// TwinCAT 3 PLC project Crane_Control
// ProgramVersion: 3.1.4026.20
// libraries:
//   Tc2_Standard, * (Beckhoff Automation GmbH)
//   Tc2_System, * (Beckhoff Automation GmbH)
// project tree:
//   Enumeration/ E_Mode.TcDUT (not stored), E_Motion.TcDUT (not stored)
//   Function Blocks/ FB_AutoClock.TcPOU, FB_ControlSignal.TcPOU, FB_Derivator.TcPOU (not stored), FB_FeedForward.TcPOU, FB_FeedForward_NonLinear.TcPOU, FB_Filtering.TcPOU, FB_Home.TcPOU, FB_InitialPos.TcPOU, FB_Integrator.TcPOU, FB_JoystickInputScaling.TcPOU, FB_KvFF.TcPOU (not stored), FB_MotionRef.TcPOU, FB_NaiveFF.TcPOU, FB_Normalize.TcPOU (not stored), FB_PID.TcPOU, FB_PositionInputScaling.TcPOU (not stored), FB_PressureFeedback.TcPOU, FB_RunClock.TcPOU (not stored), FB_Running.TcPOU, FB_ValveOutput.TcPOU (not stored)
//   Global Variable Lists/ G_Enables.TcGVL, G_FilterConstants.TcGVL (not stored), G_Filtered.TcGVL (not stored), G_Init.TcGVL, G_Inputs.TcGVL (not stored), G_Mode.TcGVL (not stored), G_OPC.TcGVL, G_Output.TcGVL, G_Parameter.TcGVL
//   / PlcTask.TcTTO
//   Programs/ MAIN.TcPOU, P_Modes.TcPOU, P_Output.TcPOU, P_RunClock.TcPOU (not stored)
// real-time tasks:
//   TASK PlcTask: cycle T#1ms, priority 20, ADS port 350
// I/O:
//   DEVICE Device 1 (EtherCAT), AmsNetId 192.168.0.204.4.1
//     RIO (EK1100) [EK1100 EtherCAT Coupler (2A E-Bus)]
//       DI (EL1008) [EL1008 8Ch. Dig. Input 24V, 3ms]
//       DO (EL2008) [EL2008 8Ch. Dig. Output 24V, 0.5A]
//       AI1 (EL3068) [EL3068 8Ch. Ana. Input 0-10V]
//       AI2 (EL3068) [EL3068 8Ch. Ana. Input 0-10V]
//       AI3 (EL3174) [EL3174 4Ch. Ana. Input +/-10V Diff., +/-20mA SingleEnded, 16 Bit]
//       AO (EL4104) [EL4104 4Ch. Ana. Output 0-10V, 16bit]
//       End Cap (EL9011) [EL9011 End Terminal]
// variable links:
//   Crane_Control/Crane_Control Instance <-> Device 1 (EtherCAT)/RIO (EK1100)/AI2 (EL3068)
//     PlcTask Inputs/G_Inputs.nRawPs <-> AI Standard Channel 1/Value

CONFIGURATION Crane_Control
    RESOURCE PLC ON TwinCAT3
        TASK PlcTask(INTERVAL := T#10ms, PRIORITY := 20);
        PROGRAM MAIN WITH PlcTask : MAIN;
    END_RESOURCE
END_CONFIGURATION

// ---- Global Variable Lists/G_Enables.TcGVL
{attribute 'qualified_only'}
// BOOL: True/False

VAR_GLOBAL
	
	// Control Enables
	bEnablePID 		: BOOL; // Enable PID Control
	bEnableFF 		: BOOL; // Enable FeedForward	
	bEnablePFB		: BOOL; // Enable Pressure Feedback
	bEnableU 		: BOOL; // Enable Signal to Valve

	bCharTesting	: BOOL; // Enable Characteristic testing
	bMove2Home		: BOOL; // Enable Home-function
	
	// No Function
	bEnableComp 	: BOOL; // Driving with Compensator
	
	// Enumerators
	nModeSelect		: E_Motion; // Motion Reference
	
END_VAR

// ---- Global Variable Lists/G_Init.TcGVL
// SINT: Integer [-128, 127]
VAR_GLOBAL CONSTANT
	SS_INITIALIZE: SINT := 0; 	// Initial system state value
	SS_STEP: SINT := 1;			// Step sequence state value
END_VAR

// ---- Global Variable Lists/G_OPC.TcGVL
{attribute 'qualified_only'}
// LREAL: Long Real decimal number

VAR_GLOBAL
	
	// Unfiltered Pressures
	fPa 				: LREAL; // [bar], Pressure A 
	fPb 				: LREAL; // [bar], Pressure B 
	fPs 				: LREAL; // [bar], Pressure Supply 
	fPaLower 			: LREAL; // [bar], Pressure A between DCV and CBV 
	
	// Filtered Pressures
	fPaFiltered 		: LREAL; // [bar], Pressure A Filtered 
	fPbFiltered 		: LREAL; // [bar], Pressure B Filtered
	fPsFiltered 		: LREAL; // [bar], Pressure Supply Filtered
	fPaLowerFiltered 	: LREAL; // [bar], Pressure A between DCV and CBV Filtered
	
	fSpoolPosition 		: LREAL; // [-1,1], Spool position
	fPistonPosition 	: LREAL; // [m], Piston position
	fPistonPosMeasured 	: LREAL; // [m], Measured piston position
	fJoystick 			: LREAL; // [-1,1], Joystick signal
	fFlow 				: LREAL; // [L/min], Flow rod-side 
	fFlowCalc 			: LREAL; // [L/min], Calculated flow
	
	fXRef 				: LREAL; // [m], Position reference [m]
	fXDotRef 			: LREAL; // [m/s], Velocity reference [m/s]
	fFlowRef 			: LREAL; // [L/min], Flow reference calculated form fXDotRef
	
	fFFFlow				: LREAL; // [L/min], Flow form feed forward
	fKv					: LREAL; // Capacity factor (how much liquid a valve can let through over a set pressure drop)

	fWantedSpoolPos 	: LREAL; // [-1,1], Wanted spool position
	fUpfbGrad 			: LREAL; // Pressure feedback gradient
	fPxGrad 			: LREAL; // Pressure gradient
	fUTest 				: LREAL; // [-1,1], Signal to Valve with pfb (pressure feedback)
	fTime 				: LREAL; // [s], Time
	fError 				: LREAL; // [m], Error
	
	
	fSignalPID 			: LREAL; // PID signal value
	fFF 				: LREAL; // FF signal Value
	fUpfb 				: LREAL; // Pressure feedback signal
	fU 					: LREAL; // [-1,1], Signal to set spool at wanted position 

END_VAR

// ---- Global Variable Lists/G_Output.TcGVL
{attribute 'qualified_only'} // Variable needs to be used with GVL-name

// INT: [-32768, 32767]	
// BOOL: True/False
// %Q* assigns next available memory adress in Twincat (Out)

VAR_GLOBAL
	// Digital Outputs
	bGreenLight 			AT %Q* : BOOL;	// Green light on controller
	bRedLight 				AT %Q* : BOOL;	// Red light on controller
	
	// Analog Outputs
	nValveOutput 			AT %Q* : INT;	// Valve output
	bRunning				AT %Q* : BOOL;
END_VAR

// ---- Global Variable Lists/G_Parameter.TcGVL
{attribute 'qualified_only'}
// LREAL: Long Real decimal number
// INT: [-32768, 32767]	

VAR_GLOBAL
	// Motion Ref
	// Sine Parameters
	fAmplitude 		: LREAL := 0.15;
	fMean 			: LREAL := 0.2;
	fFrequency 		: LREAL := 0.05;
	
	
	// Valve Values
	// Flow
	fQMaxDown 		: LREAL := 10.0; // [L/min]
	fQMaxUp 		: LREAL := 10.0; // [L/min]	
	
	// Area
	fAreaUp 		: LREAL := 33.100/1E4; //[m^2]
	fAreaDown 		: LREAL := 23.560/1E4; //[m^2]
	
	// Deadband
	fDeadUp 		: LREAL := 0.23;
	fDeadDown 		: LREAL := 0.215;
	
	fMaxSpeed 		: LREAL := 0.01; // [m/s] 
	fDeltaP0 		: LREAL := 8.0; // [Bar]
	
	// Deadband test
	fConst 			: LREAL := 0.0; // [-1, 1]

	fCycleTime 		: LREAL := 0.001; // Time Step [s]
	fQConst 		: LREAL := 15;
	fPistonStroke 	: LREAL := 0.5;
	
	// PID-constants
	Kp 				: LREAL := 14.0; 	// P
	Ki 				: LREAL := 0.0;		// I
	Kd 				: LREAL := 0.0;		// D
	
	// Pressure feedback constants
	Kf				: LREAL := 2E-4;
	TauF			: LREAL := 0.1; // [0.05 .. 0.1]
	PFBstate		: INT 	:= 2; // 0:Switching, 1: Pa-phi*Pb, 2: Pb
	FFMode			: INT 	:= 1; // 0: Bachelor FF, 1: Kv FF, 2: Naive FF

END_VAR

// ---- Programs/MAIN.TcPOU
PROGRAM MAIN
VAR
END_VAR

P_Inputs();
P_Filtering();
P_ControlBlock();
P_Output();
//P_RunClock();
P_Modes();
P_PID();
P_FeedForward();

END_PROGRAM

// ---- Programs/P_Output.TcPOU
PROGRAM P_Output

VAR
	fbValveOutput : FB_ValveOutput;
END_VAR

// Runs FB with given values
fbValveOutput(
	fNormalizedInput := G_OPC.fU,
	bEnable := G_Enables.bEnableU,
	nOutput => G_Output.nValveOutput	
);

IF G_Mode.bRunning THEN // If system is running, set green and red light on controller true. False when not running
	G_Output.bGreenLight := TRUE;
	G_Output.bRedLight := TRUE;
ELSE
	G_Output.bGreenLight := FALSE;
	G_Output.bRedLight := FALSE;
END_IF

END_PROGRAM

// ---- Programs/P_Modes.TcPOU
PROGRAM P_Modes

VAR
	fbRunning : FB_Running;
END_VAR

// Runs FB with given values
fbRunning(
	bAuto := G_Inputs.bAuto, 			// Auto mode controller
	bManual := G_Inputs.bManual, 		// Manual mode controller
	bStart := G_Inputs.bStartButton,	// Start button
	bStop := G_Inputs.bStopButton, 		// Stop button
	
	// Values from FB sent to GVL
	bRunning => G_Mode.bRunning,
	bRunning => G_Output.bRunning,
	bManualMode => G_Mode.bManual,
	bAutoMode => G_Mode.bAuto
);

END_PROGRAM

// ---- Function Blocks/FB_Running.TcPOU
FUNCTION_BLOCK FB_Running
// BOOL: True/False

// Input variables
VAR_INPUT
	bManual : BOOL;
	bStart : BOOL;
	bStop : BOOL;
	bAuto : BOOL;
END_VAR

// Output variables
VAR_OUTPUT
	bRunning : BOOL;
	bAutoMode : BOOL;
	bManualMode : BOOL;
END_VAR


IF NOT(bStart) AND NOT(bManual) AND NOT(bAuto) OR (bStop) THEN // If nothing active, all false values
	bRunning := FALSE;
	bAutoMode := FALSE;
	bManualMode := FALSE;	
	
ELSIF bStart AND bAuto AND NOT(bStop) THEN // If start button and auto is true (auto mode)
	bRunning := TRUE;
	bAutoMode := TRUE;
	bManualMode := FALSE;
	
ELSIF bStart AND bManual AND NOT(bStop) THEN // If start and manual is true (manual mode)
	bRunning := TRUE;
	bManualMode := TRUE;
	bAutoMode := FALSE;
END_IF

END_FUNCTION_BLOCK

// ---- Function Blocks/FB_AutoClock.TcPOU
FUNCTION_BLOCK FB_AutoClock
// LREAL: Long Real decimal number
// BOOL: True/False

// Input variables
VAR_INPUT
	fStart : BOOL; // Start timer
	fRunning : BOOL; // System is running
	fCycle : LREAL; // Time step
END_VAR

// Output variables
VAR_OUTPUT
	fTime : LREAL; // Output (time)
END_VAR


IF NOT(fStart) OR NOT(fRunning) THEN // If start signal is missing or the system is not running, set time to zero
	fTime := 0.0; 
ELSIF fStart AND fRunning THEN // If both start signal and system is on. PLS ticks synced into real time
	fTime := fTime + fCycle;		
END_IF

END_FUNCTION_BLOCK

// ---- Function Blocks/FB_ControlSignal.TcPOU
FUNCTION_BLOCK FB_ControlSignal
// LREAL: Long Real decimal number
// INT: [-32768, 32767]	
// BOOL: True/False

// Input variables
VAR_INPUT
	fFF 			: LREAL; // FF signal value
	fPID			: LREAL; // PID signal value
	fPFB			: LREAL; // Pressure feedback signal
	
	// Deadband
	fDeadBandUp		: LREAL; 
	fDeadBandDown	: LREAL;
	
	nFFState		: INT; // 0: Bachelor FF, 1: Kv FF, 2: Naive FF

	bPID			: BOOL; // Enable PID control
	bFF				: BOOL; // Enable feed forward
	bPFB			: BOOL; // Enable pressure feedback
	bU				: BOOL; 
	bValve			: BOOL; 
END_VAR

// Output variables
VAR_OUTPUT
	fU				: LREAL; // Final output
	fUAdj			: LREAL; // Adjusted signal before final output
END_VAR

// Variables
VAR
	FF				: LREAL; // Feed forward
	PID				: LREAL; // PID
	PFB				: LREAL; // Pressure feedback
END_VAR


FF := fFF  * TO_INT(bFF); // Multiplies fFF with bFF. bFF:(True/False) = (1/0). Like an on/off switch for the feed forward.

PID := fPID * TO_INT(bPID); // On/off switch for PID

PFB := fPFB * TO_INT(bPFB); // On/off switch for pressure feedback

fUAdj := (FF+PID-PFB)*TO_INT(bValve); // bValve works as a main on/off switch

IF FF = 0.0 THEN // If feed forward is off
	fU := 0.0; // Output = 0
ELSE
	CASE nFFState OF // Feed forward states 0,1,2
		0: // State 0
			IF (fUAdj > 0.0) THEN
				fU := fUAdj + fDeadBandUp; // Adds offset to skip deadband in the valve (positive direction)
			ELSIF (fUAdj < 0.0) THEN
				fU := fUAdj - fDeadBandDown; // Adds offset to skip deadband in the valve (negative direction)
			ELSE
				fU := 0.0;
			END_IF
			
		ELSE // FF States that use this: 1, 2
			IF (fUAdj > 0.0) THEN
				fU := fUAdj;
			ELSIF (fUAdj < 0.0) THEN
				fU := fUAdj;
			ELSE
				fU := 0.0;
			END_IF
	END_CASE
END_IF

// Saturation for output [-1,1]
IF fU < -1.0 THEN
	fU := -1.0; 
ELSIF fU > 1.0 THEN
	fU := 1.0;
ELSE
	fU := fU;
END_IF

END_FUNCTION_BLOCK

// ---- Function Blocks/FB_FeedForward.TcPOU
FUNCTION_BLOCK FB_FeedForward
// LREAL: Long Real decimal number

// Input variables
VAR_INPUT
	fXDotRef 		: LREAL; // Velocity Reference [m/s]
	fMaxFlowUp 		: LREAL; // Needs to be positive (22)
	fMaxFlowDown 	: LREAL; // Needs to be positive (15)
	fDeadUp			: LREAL; // Needs to be positive (0.155)
	fDeadDown 		: LREAL; // Needs to be positive (0.18)
	
	fPs 			: LREAL; // [Bar]
	fPa 			: LREAL; // [Bar]
	fPb 			: LREAL; // [Bar]
	fDeltaP0		: LREAL; // [Bar] (8.0)
	fAreaUp			: LREAL; // [mm^2]
	fAreaDown		: LREAL; // [mm^2]
END_VAR

// Output variables
VAR_OUTPUT
	fUFF 			: LREAL;	// FF signal value
	fFlow			: LREAL; 	// Wanted Flow
	fFlowLM			: LREAL;	// Flow [L/min]
END_VAR

// Variables
VAR
	fDeltaP_Norm	: LREAL; 	// Pressure Drop with Compensator
	
	fDeltaP			: LREAL; 	// Pressure Drop
	fDeltaP_Ref		: LREAL; 	// Reference Pressure Drop
	fFlowRef		: LREAL; 	// Reference Flow
	
	fUFFTemp		: LREAL;	// Temp Signal Out
END_VAR


fDeltaP_Norm	:= fDeltaP0 * 100000.0; // Converts from bar to Pa

IF fXDotRef > 0.0 THEN // Velocity reference > 0
	fFlow := fXDotRef * fAreaUp; // Calculates wanted flow (Q = v*A)
	fFlowLM := -fFlow * 60000; // Converts flow to [L/min]. Negative sign for valve direction
	fDeltaP := (fPs - fPa) * 100000.0; // Calculates pressure drop
	
	IF fDeltaP < 100 THEN // Safety for pressure drop to never go below 100. Avoiding division by zero
		fDeltaP := 100;
	ELSE
		fDeltaP := fDeltaP;
	END_IF
	
	fDeltaP_Ref := ABS(fDeltaP_Norm/ (fDeltaP)); // Calculates reference pressure drop. 
	fFlowRef := (fFlow * SQRT(fDeltaP_Ref)) * 60000.0; // Calculates reference flow
	fUFFTemp := fFlowRef/fMaxFlowUp; // Normalizes output signal [0,1]
	fUFFTemp := -fUFFTemp * (1.0-fDeadUp); // Adjusts for valve deadband 
	
ELSIF fXDotRef < 0.0 THEN // Velocity reference < 0
	fFlow := fXDotRef * fAreaDown; // Calculates wanted flow (Q = v*A)
	fFlowLM := -fFlow * 60000; // Converts flow to [L/min]. Negative sign for valve direction
	fDeltaP := (fPs - fPb) * 100000.0; // Calculates pressure drop
	
	IF fDeltaP < 100 THEN // Safety for pressure drop to never go below 100. Avoiding division by zero
		fDeltaP := 100;
	ELSE
		fDeltaP := fDeltaP;
	END_IF
	
	fDeltaP_Ref := ABS(fDeltaP_Norm/(fDeltaP)); // Calculates reference pressure drop
	fFlowRef := (fFlow * SQRT(fDeltaP_Ref)) * 60000.0; // Calculates reference flow
	fUFFTemp := fFlowRef/fMaxFlowDown; // Normalizes output signal [-1,0]
	fUFFTemp := -fUFFTemp*(1.0-fDeadDown); // Adjusts for valve deadband
	
ELSE
	
	fUFFTemp := 0.0; // FF signal is zero		

END_IF

// Safety to keep FF signal [-1,1]
IF fUFFTemp > 1.0 THEN
	fUFF := 1.0;
ELSIF fUFFTemp < -1.0 THEN
	fUFF := -1.0;
ELSE
	fUFF := fUFFTemp;
END_IF

END_FUNCTION_BLOCK

// ---- Function Blocks/FB_FeedForward_NonLinear.TcPOU
FUNCTION_BLOCK FB_FeedForward_NonLinear
// LREAL: Long Real decimal number

// Input variables
VAR_INPUT
	fXDotRef 		: LREAL; // Velocity Reference [m/s]
	fMaxFlowUp 		: LREAL; // Needs to be positive (22)
	fMaxFlowDown 	: LREAL; // Needs to be positive (15)
	fDeadUp			: LREAL; // Needs to be positive (0.155)
	fDeadDown 		: LREAL; // Needs to be positive (0.18)

	fPs 			: LREAL; // [Bar]
	fPa 			: LREAL; // [Bar]
	fPb 			: LREAL; // [Bar]
	fDeltaP0		: LREAL; // [Bar]
	fAreaUp			: LREAL; // [mm^2]
	fAreaDown		: LREAL; // [mm^2]
END_VAR

// Output variables
VAR_OUTPUT
	fUFF 			: LREAL;	// FF signal value
	fFlow			: LREAL; 	// Wanted Flow
	fFlowLM			: LREAL;	// Flow [L/min]
END_VAR

// Variables
VAR
	fDeltaP_Norm	: LREAL; 	// Pressure Drop with Compensator
	
	fDeltaP			: LREAL; 	// Pressure Drop
	fDeltaP_Ref		: LREAL; 	// Reference Pressure Drop
	fFlowRef		: LREAL; 	// Reference Flow
	
	fUFFTemp		: LREAL;	// Temp Signal Out
END_VAR

// Non-linear FF compensates for disturbances where the relationship is not proportional/constant. 

fDeltaP_Norm	:= fDeltaP0 * 100000.0; // Converts from bar to Pa

IF fXDotRef > 0.0 THEN // If velocity reference > 0
	
	fFlow := fXDotRef * fAreaUp; // Calculates wanted flow 
	fFlowLM := -fFlow * 60000; // Converts flow to [L/min]. Negative sign for valve direction
	fDeltaP := (fPs - fPa) * 100000.0; // Calculates pressure drop
	IF fDeltaP < 100 THEN // Safety for pressure drop to never go below 100. Avoiding division by zero
		fDeltaP := 100;
	ELSE
		fDeltaP := fDeltaP;
	END_IF
	fDeltaP_Ref := ABS(fDeltaP_Norm/ (fDeltaP)); // Calculates reference pressure drop
	fFlowRef := (fFlow * SQRT(fDeltaP_Ref)) * 60000.0; // Calculates reference flow
	fUFFTemp := fFlowRef/fMaxFlowUp; // Normalizes output signal [0,1]
	fUFFTemp := -fUFFTemp * (1.0-fDeadUp); // Adjusts for valve deadband
	
ELSIF fXDotRef < 0.0 THEN
	
	fFlow := fXDotRef * fAreaDown;
	fFlowLM := -fFlow * 60000;
	fDeltaP := (fPs - fPb) * 100000.0;
	IF fDeltaP < 100 THEN
		fDeltaP := 100;
	ELSE
		fDeltaP := fDeltaP;
	END_IF
	fDeltaP_Ref := ABS(fDeltaP_Norm/(fDeltaP));
	fFlowRef := (fFlow * SQRT(fDeltaP_Ref)) * 60000.0;
	fUFFTemp := fFlowRef/fMaxFlowDown; 
	fUFFTemp := -fUFFTemp*(1.0-fDeadDown);
	
ELSE
	
	fUFFTemp := 0.0;		

END_IF

IF fUFFTemp > 1.0 THEN
	fUFF := 1.0;
ELSIF fUFFTemp < -1.0 THEN
	fUFF := -1.0;
ELSE
	fUFF := fUFFTemp;
END_IF

END_FUNCTION_BLOCK

// ---- Function Blocks/FB_Filtering.TcPOU
FUNCTION_BLOCK FB_Filtering
// SINT: Integer [-128, 127]
// LREAL: Long Real decimal number
// USINT: Integer, strictly positive [0,255]

// Input variables
VAR_INPUT
	ssMethodType: SINT;
	Signal: LREAL; 	// Input signal
	Num: LREAL; 	// Filter constant
	DenZ: LREAL; 	// Filter constant
	Den: LREAL; 	// Filter constant
	Initial: LREAL; // Filter constant
END_VAR

// Output variables
VAR_OUTPUT
	Signal_Unfiltered: LREAL;	// Unfiltered signal
	Signal_Filtered: LREAL;		// Filtered signal
END_VAR

// Variables
VAR
	DiscreteTransferFcn1_icLoad: USINT; // Initial condition load (start value)
	DiscreteTransferFcn1_states: LREAL; // Filter state/memory (how the filter works)
	c_TmpSignalConversionAtDisc: ARRAY[0..1] OF LREAL; // List of two decimal numbers
END_VAR



CASE ssMethodType OF
    SS_INITIALIZE: // If ssMethodType = SS_INITIALIZE, set initial condition load = 1.
        DiscreteTransferFcn1_icLoad := 1;
    SS_STEP: // If ssMethodType = SS_STEP, set filter constants
        c_TmpSignalConversionAtDisc[0] := DenZ;
        c_TmpSignalConversionAtDisc[1] := Den;
		
        IF DiscreteTransferFcn1_icLoad <> 0 THEN // If icLoad is not equal to zero, set initial filter value
            DiscreteTransferFcn1_states := Initial;
        END_IF;
        Signal_Filtered := Num * DiscreteTransferFcn1_states; // Output = filter constant * filter state
        Signal_Unfiltered := Signal;
        DiscreteTransferFcn1_icLoad := 0; // Reset filter initial condition
        DiscreteTransferFcn1_states := Signal - (c_TmpSignalConversionAtDisc[1] * DiscreteTransferFcn1_states); // Filter update (negative feedback)
END_CASE;

END_FUNCTION_BLOCK

// ---- Function Blocks/FB_Home.TcPOU
FUNCTION_BLOCK FB_Home
// LREAL: Long Real decimal number
// BOOL: True/False

// Input variables
VAR_INPUT
	bGoHome : BOOL; // Enable home function
	fCurrentPos : LREAL; // Piston position [m]
	fTolerance : LREAL; // Tolerance for position [m]
	fMoveTime : LREAL; // set to 10[s]
	fHomePos : LREAL; // set to 0.05 (10%) [m]
	fMoveTimer : LREAL; // Timer [s]
END_VAR

// Output variables
VAR_OUTPUT
	fXRef : LREAL; // Position reference [m]
	fXDotRef : LREAL; // Velocity reference [m/s]
END_VAR




IF bGoHome AND ABS(fHomePos-fCurrentPos)>fTolerance THEN // If home command is active and distance to home is larger than allowed tolerance
	fXDotRef := (fHomePos-fCurrentPos)/fMoveTime; // Calculates speed
	fXRef := fCurrentPos + fXDotRef * fMoveTimer; // Calculates position
	IF	ABS(fHomePos-fCurrentPos)<=fTolerance THEN // If distance is lower than allowed tolerance, home position is aquired
		bGoHome := FALSE;
		fXDotRef := 0.0;
		fXRef := fCurrentPos;
	END_IF
ELSE // Stop moving and stay at current position
	fXDotRef := 0.0;
	fXRef := fCurrentPos;
END_IF

END_FUNCTION_BLOCK

// ---- Function Blocks/FB_InitialPos.TcPOU
FUNCTION_BLOCK FB_InitialPos
// LREAL: Long Real decimal number
// BOOL: True/False

// Input variables
VAR_INPUT
	bEnable : BOOL; // Start signal on controller
	fCurrentPos : LREAL; // Piston position [m]
END_VAR

// Output variables
VAR_OUTPUT
	fInitialPos : LREAL; // Initial position
END_VAR

IF bEnable THEN
	fInitialPos := fInitialPos; // If system is running, keep initial position
ELSE 
	fInitialPos := fCurrentPos; // If system is off, track initial position
END_IF

END_FUNCTION_BLOCK

// ---- Function Blocks/FB_Integrator.TcPOU
FUNCTION_BLOCK FB_Integrator
// SINT: Integer [-128, 127]
// LREAL: Long Real decimal number

// Constant variables
VAR CONSTANT
	f_SampleTime: LREAL := 0.001;
END_VAR	

// Input variables
VAR_INPUT
	ssMethodType: SINT; // Integration mode (initialize or next step)
	fSignal: LREAL; 	// Signal value to integrate
END_VAR

// Output variables
VAR_OUTPUT
	fSignalIntegrated: LREAL; // Output variable after integration
END_VAR

// Variables
VAR
	c_DiscreteTimeIntegrator_DS: LREAL; // Current value/internal memory, discrete step
END_VAR

// Discrete integration

CASE ssMethodType OF 
    SS_INITIALIZE: 
        c_DiscreteTimeIntegrator_DS := 0.0; // If SS_INITIALIZE = ssMethodType -> Initialization of the integrator

    SS_STEP: 
        fSignalIntegrated := c_DiscreteTimeIntegrator_DS; // Output value = current value/internal mamory
        c_DiscreteTimeIntegrator_DS := (f_SampleTime * fSignal) + c_DiscreteTimeIntegrator_DS; // Discrete integration formula (forward euler method).
END_CASE;

END_FUNCTION_BLOCK

// ---- Function Blocks/FB_JoystickInputScaling.TcPOU
FUNCTION_BLOCK FB_JoystickInputScaling
// LREAL: Long Real decimal number
// INT: [-32768, 32767]	
// BOOL: True/False

// Input variables
VAR_INPUT
	bEnable 				: BOOL;
	nRawInput 				: INT;
	fMaxValue 				: LREAL;
	fMaxInputValue			: LREAL;
	fMinInputValue 			: LREAL;
	fNeutralInputValue  	: LREAL;
	fNeutralDeadband		: LREAL;
END_VAR

// Output variables
VAR_OUTPUT
	fOutput : LREAL;
END_VAR

// Variables
VAR
	fRawInput : LREAL;
	fTempInput : LREAL; // Temporary input
	fTempOutput : LREAL; // Temporary output

	fMaxOutputValue  		: LREAL := 1.0;
	fMinOutputValue  		: LREAL := -1.0;
	fNeutralOutputValue  	: LREAL := 0.0;
END_VAR

// Crane is only supported for movement in the y-axis (up/down)

fRawInput := INT_TO_LREAL(nRawInput); // Converts input to decimal number
fTempInput := fRawInput - fNeutralInputValue; // Defines joystick neutral point 

IF fTempInput > fNeutralDeadband THEN // Checks if joystick is moved above the neutral deadband (positive y) 
	fTempOutput := fTempInput/(fMaxInputValue - fNeutralInputValue); // Scales positive movement [0,1]
ELSIF fTempInput < -fNeutralDeadband THEN // Checks if joystick is moved below the neutral deadband (negative y)
	fTempOutput := fTempInput/(fNeutralInputValue - fMinInputValue); // Scales negative movement [-1,0]
ELSE
	fTempOutput := 0.0; // If joystick is inside deadzone, fTempOutput = 0
END_IF

IF NOT(bEnable) THEN // If bEnable is not true, set fOutput = 0
	fOutput := 0.0;
ELSE
	fOutput := LIMIT(fMinOutputValue * fMaxValue, fTempOutput * fMaxValue, fMaxOutputValue* fMaxValue); 
	// Calculates output signal within safety limits (Min, Output, Max)
END_IF

END_FUNCTION_BLOCK

// ---- Function Blocks/FB_MotionRef.TcPOU
FUNCTION_BLOCK FB_MotionRef
// LREAL: Long Real decimal number
// INT: [-32768, 32767]

// Input variables
VAR_INPUT
	fAmplitude : LREAL;		// Amplitude
	fFrequency : LREAL;		// Frequency
	fInitialPos : LREAL; 	// Initial position
	fCurrentPos : LREAL; 	// Current position
	nMotionMode : INT;		// Motion mode
	fMotionTimer : LREAL;	// Timer for movement
END_VAR

// Output variables
VAR_OUTPUT
	fXDotRef : LREAL;	 // Velocity reference
	fXRef : LREAL;		 // Position reference
	fWantedFlow : LREAL; // Flow reference calculated from velocity reference
END_VAR

// Variables
VAR
	fPI : LREAL := 3.1415;
	fMean : LREAL;
	
	arrBounduary 	: ARRAY[0..1] OF LREAL := [G_Parameter.fPistonStroke * 0.1, G_Parameter.fPistonStroke * 0.9]; // Min, Max [m]
	// arrBounduary[0] and arrBoundary[1] = Lower limit piston stroke (10%) and higher limit (90%) of 0.5m. Safety for cylinder movement
	
	fRampTime 	 	: LREAL := 15.0; // [s] duration of movement sequence in ramp mode. Cylinder uses 15s from 10% to 90%
 	fTolerance   	: REAL := 0.005;  // ±5 mm tolerance for cylinder 
  	
END_VAR




CASE nMotionMode OF
	0:	// Sine 
		fMean := fAmplitude + fInitialPos; // Midpoint of the sine-wave. Initial position +- 0.15m
		fXRef := fMean - fAmplitude * COS(2*fPI * fFrequency * fMotionTimer); // Position ref. Angle calculated using a timer, cylinder starts going upwards
		fXDotRef := 2 * fPI *fFrequency * fAmplitude * SIN(2*fPI * fFrequency * fMotionTimer); // Velocity ref. Position derivated
		
	1:	// Ramp
		IF fMotionTimer <= fRampTime THEN // If motion timer < 15s
			fXDotRef := (arrBounduary[1] - arrBounduary[0]) / fRampTime; //calculates speed: distance/time = (90%-10%)/ramp time
			fXRef := arrBounduary[0] + fXDotRef * fMotionTimer; // position = velocity*time = 10% + speed*time (10%: start distance)
			
		ELSIF fMotionTimer <= fRampTime * (4.0/3.0) THEN // If motion timer < 20s
			fXRef := arrBounduary[1]; // Position holds at 90% (Highest position)
			fXDotRef := 0.0; // Velocity = 0
			
		ELSIF fMotionTimer <= (2.0 + 1.0/3.0) * fRampTime AND fMotionTimer > fRampTime * (4.0/3.0) THEN // If motion timer is [20,35]s
			fXDotRef := (arrBounduary[0] - arrBounduary[1]) / fRampTime; // Velocity = (10%-90%)/ramp time. Cylinder retracting
			fXRef := arrBounduary[1] + fXDotRef * (fMotionTimer - (4.0/3.0) * fRampTime); 
			// position = velocity*time = 90% + speed*time (90%: start distance). Timer calculated to start at 0 on the top position where motion timer = 20s
		
		ELSIF fMotionTimer > (2.0 + 1.0/3.0) * fRampTime THEN // If timer > 35
			fXDotRef := 0.0; // Velocity = 0
			fXRef := arrBounduary[0]; // Position holds at 10% (Lowest position)
		END_IF
END_CASE

IF fXDotRef > 0.0 THEN // If cylinder moves upwards
	fWantedFlow := fXDotRef * G_Parameter.fAreaUp*6E4; // Wanted flow = speed * AreaUp
ELSIF fXDotRef < 0.0 THEN // If cylinder moves downwards
	fWantedFlow := fXDotRef * G_Parameter.fAreaDown*6E4; // Wanted flow = speed * AreaDown
ELSE
	fWantedFlow := 0.0; 
END_IF

END_FUNCTION_BLOCK

// ---- Function Blocks/FB_NaiveFF.TcPOU
FUNCTION_BLOCK FB_NaiveFF
// LREAL: Long Real decimal number

// Input variables
VAR_INPUT
	fPs 		: LREAL; // [bar] Pressur supply
	fPa 		: LREAL; // [bar] Pressure A between DCV and CBV 
	fPb 		: LREAL; // [bar] Pressure B
	
	fXDotRef 	: LREAL; // [m/s] Velocity reference
END_VAR

// Output variables
VAR_OUTPUT
	fFF 		: LREAL; // [-1,1], Feed forward signal value (spool position)
	fFlow 		: LREAL; // [L/min] Feed forward flow output
	fKv 		: LREAL; // [L/min / bar^0.5] Capacity factor
END_VAR

// Variables
VAR
	fDeltaP		: LREAL; // [bar] pressure drop
END_VAR

// Naive FF assumes relationship between in/out is linear. 
// Multiplies input with a fixed gain to estimate the output.

IF fXDotRef > 0.0 THEN  // When cylinder velocity REFERENCE > 0
	fFlow := fXDotRef * G_Parameter.fAreaUp * 6E4; // Calculates needed flow (Q = v*A)
	fDeltaP := fPs - fPa; // Calculates pressure drop over valve
	
	fFF := -(0.2143 + 0.7857 * fKv/3.7796); // Calculates signal value (spool position)
ELSIF fXDotRef < 0.0 THEN // When cylinder velocity REFERENCE < 0
	fFlow := fXDotRef * G_Parameter.fAreaDown * 6E4; // Calculates needed flow (Q = v*A)
	fDeltaP := fPs - fPb; // Calculates pressure drop over valve
	
	fFF := (0.2143 + 0.7857 * fKv/3.7796); // Calculates signal value (spool position)
ELSE
	fFlow := 0.0;
	fFF := 0.0;
END_IF

IF fDeltaP <= 0.0 THEN // If pressure in is lower than in the cylinder
	fKv := 4.0; // Capacity factor
ELSE
	fKv := ABS(fFlow)/SQRT(fDeltaP); // Capacity factor else
END_IF

END_FUNCTION_BLOCK

// ---- Function Blocks/FB_PID.TcPOU
FUNCTION_BLOCK FB_PID
// LREAL: Long Real decimal number
// BOOL: True/False

// Input variables
VAR_INPUT
	bEnablePID			: BOOL;  // Enables PID controller
	fX 					: LREAL; // Position reference [m]
	fXReal 				: LREAL; // Piston position [m]
	fSignalIntegrated 	: LREAL; // Integrated signal
	fSignalDerivated 	: LREAL; // Derivated signal
	fKp 				: LREAL; // P constant
	fKi 				: LREAL; // I constant
	fKd 				: LREAL; // D constant
END_VAR

// Output variables
VAR_OUTPUT
	fSignalI 			: LREAL;
	fSignalD 			: LREAL;
	fSignalAdjusted 	: LREAL; // PID signal value
	fError  			: LREAL; // Error
END_VAR

// Variables
VAR
	fTempP 				: LREAL; // Temporary P value
	fTempI 				: LREAL; // Temporary I value
	fTempD 				: LREAL; // Temporary D value
	fTempOut 			: LREAL; // Temporary output
END_VAR

fError := fX - fXReal; // Position error

fSignalI := fError; 
fSignalD := fError; 

fTempP := fError * fKp; // Calculates proportional term (current error)
fTempI := fSignalIntegrated * fKi; // Calculates integral term (past error)
fTempD := fSignalDerivated * fKd; // Calculates derivator term (future trend)

fTempOut := -(fTempP + fTempI + fTempD); // PID-controller (minus sign for correct cylinder movement)

IF fTempOut > 1.0 THEN
	fSignalAdjusted := 1.0; // Max-saturation
ELSIF fTempOut < -1.0 THEN
	fSignalAdjusted := -1.0; // Min-saturation
ELSE
	fSignalAdjusted := fTempOut; // PID-signal
END_IF

// Safety switch
IF bEnablePID THEN
	fSignalAdjusted := fSignalAdjusted;
ELSE
	fSignalAdjusted := 0.0;
END_IF

END_FUNCTION_BLOCK

// ---- Function Blocks/FB_PressureFeedback.TcPOU
FUNCTION_BLOCK FB_PressureFeedback
// INT: [-32768, 32767]	
// LREAL: Long Real decimal number

// Input variables
VAR_INPUT
	fKf			: LREAL; // Pressure feedback constant
	fTauF		: LREAL; // Pressure feedback constant [s]	
	state		: INT;	 // [0,1,2] 0:Switching, 1: Pa-phi*Pb, 2: Pb
END_VAR

// Output variables
VAR_OUTPUT
	fUpfb 		: LREAL; // Pressure feedback signal
	fUpfbGrad	: LREAL; // Pressure feedback gradient
	fPxGrad		: LREAL; // Pressure gradient [Bar]
END_VAR

// Variables
VAR
	fDt			: LREAL := 0.001; // Delta time [s]
	fPx			: LREAL := 0.0; // Pressure [Bar]
	fPxOld		: LREAL; // Previous pressure[Bar]
	fARatio		: LREAL; // Valve area ratio
END_VAR


CASE state OF
	0: // Altering input for Px (switching state)
		IF G_OPC.fU < 0.0 THEN // If signal to set spool at wanted position [-1,1] is < 0: pressure = pressure A
			fPx := G_OPC.fPa;
		ELSIF G_OPC.fU > 0.0 THEN // If signal to set spool at wanted position [-1,1] is > 0: pressure = pressure B
			fPx := G_OPC.fPb;
		ELSE
			fPx := 0.0; 
		END_IF
	1:	// Px = Pa - phi * Pb
		fARatio := G_Parameter.fAreaDown/G_Parameter.fAreaUp; // Area ratio = AreaDown/AreaUp
		fPx := G_OPC.fPa - fARatio * G_OPC.fPb;  // Effective pressure = pA-pB. Uses area ratio to get equivalent pressure
	2:	// Px = Pb
		fPx := G_OPC.fPb;
END_CASE

fPxGrad := (fPx - fPxOld)/fDt; // Change of pressure per second (this instant)
fUpfbGrad :=  (fKf * fPxGrad - fUpfb)/fTauF; // Change of pressure (filtered/overall)
fUpfb := fUpfb + fUpfbGrad * fDt; // Updates pressure feedback (Eulers method)

fPxOld := fPx; // Updates previous pressure

END_FUNCTION_BLOCK
